FUNCTION_BLOCK FB_Lamp
VAR_INPUT
END_VAR
VAR_OUTPUT
END_VAR
VAR
	_nPowerConsumption	: UDINT := 1234;
END_VAR

PROPERTY nPowerConsumption : UDINT
GET
nPowerConsumption := _nPowerConsumption;
END_GET
END_PROPERTY

END_FUNCTION_BLOCK

(* stored: Version 1.1.0.1, ProductVersion 3.1.4024.12
   POU FB_Lamp: Id {d4c89d15-b770-45c8-b729-af82b526254a}, SpecialFunc None
   Property nPowerConsumption: Id {1fe18b4a-5755-4893-8591-56a3b6f7f5c9}
   Get Get: Id {2f81a754-0162-489e-af33-00e731e88eed} *)
